# EPICS IOC start-up script: iocsh/ethercatmcAxisdebug-twincat-ads.iocsh
dbLoadRecords("ethercatmcdebug-twincat-ads.template", "SYSPFX=$(SYSPFX), AXIS_NAME=$(AXIS_NAME), ASYN_PORT=$(ASYN_PORT), MOTOR_PORT=$(MOTOR_PORT), AXIS_NO=$(AXIS_NO), PREC=3")
